TYPE AdditionalService_Struct :
UNION
		Value : INT;
		Bits : Bits_CommonBlock;
END_UNION
END_TYPE

(* stored: Version 1.1.0.1, ProductVersion 3.1.4024.2
   DUT AdditionalService_Struct: Id {738fd2ab-0d04-44ce-9583-2a9c22e19046} *)
